{attribute 'qualified_only'}
VAR_GLOBAL
	g_motionTest 	: ST_PTMotionTest;
	g_cycleTest 	: ST_PTCycleTest;
	g_caliData 		: ST_PTCaliData;
END_VAR

(* stored: Version 1.1.0.1, ProductVersion 3.1.4024.11
   GVL GVL_PTInstruction: Id {0e07da42-d08b-4b00-b116-9e59ec443a45} *)
